FUNCTION_BLOCK FBlock (* Basic function block *)
  (* Standard: 61499 *)
  (* Version 1.0, 11/20/2015 9:00 AM, Kawsihen, Kawsihen_s Macintosh *)
  (* Compiler header: package mypackage *)
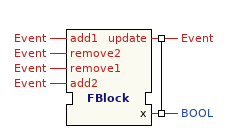
  EVENT_INPUT
    add1;
    remove2;
    remove1;
    add2;
  END_EVENT
  EVENT_OUTPUT
    update WITH x;
  END_EVENT
  VAR_OUTPUT
    x : BOOL;
  END_VAR
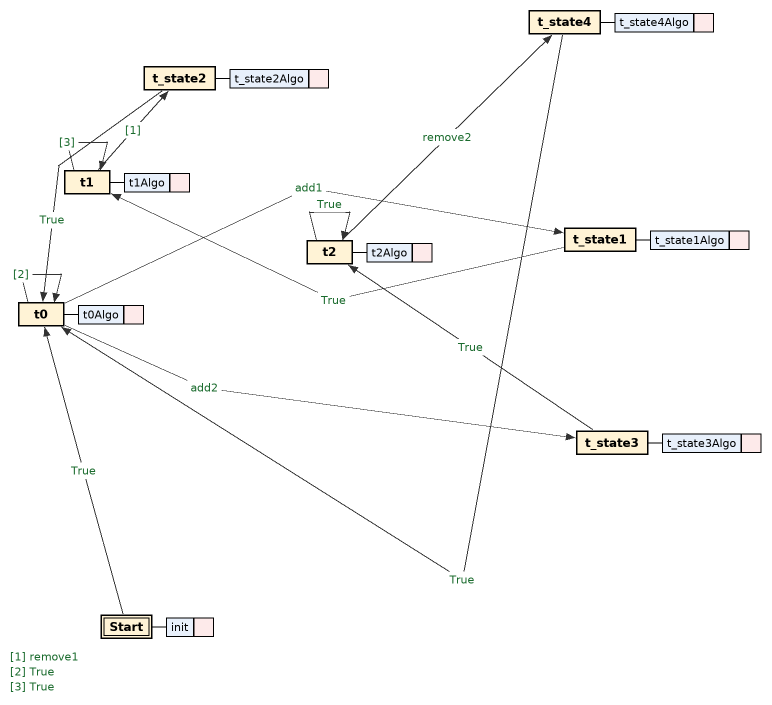
  EC_STATES
    Start : init;
    t0 : t0Algo;
    t1 : t1Algo;
    t2 : t2Algo;
    t_state1 : t_state1Algo;
    t_state2 : t_state2Algo;
    t_state3 : t_state3Algo;
    t_state4 : t_state4Algo;
  END_STATES
  EC_TRANSITIONS
    Start TO t0 := True;
    t0 TO t_state1 := add1;
    t_state1 TO t1 := True;
    t1 TO t_state2 := remove1;
    t_state2 TO t0 := True;
    t0 TO t_state3 := add2;
    t_state3 TO t2 := True;
    t2 TO t_state4 := remove2;
    t_state4 TO t0 := True;
    t0 TO t0 := True;
    t1 TO t1 := True;
    t2 TO t2 := True;
  END_TRANSITIONS
  ALGORITHM t0Algo IN C:
me->x = (float) me->C1x*exp(0.1*me->d*me->k) + 500.0;
me->k++;
  END_ALGORITHM
  ALGORITHM t1Algo IN C:
me->x = (float) me->C1x*exp(0.1*me->d*me->k) + 560.0;
me->k++;
  END_ALGORITHM
  ALGORITHM t2Algo IN C:
me->x = (float) me->C1x*exp(0.1*me->d*me->k) + 600.0;
me->k++;
  END_ALGORITHM
  ALGORITHM init IN C:
me->d = 0.01;
me->k=0;
 me->x= 510;
  END_ALGORITHM
  ALGORITHM t_state1Algo IN C:
me->x = x;
me->k = 0;
  END_ALGORITHM
  ALGORITHM t_state2Algo IN C:
me->x = x;
me->k = 0;
  END_ALGORITHM
  ALGORITHM t_state3Algo IN C:
me->x = x;
me->k = 0;
  END_ALGORITHM
  ALGORITHM t_state4Algo IN C:
me->x = x;
me->k = 0;
  END_ALGORITHM
END_FUNCTION_BLOCK
